FUNCTION_BLOCK XtsMotorModule EXTENDS CyclicBase IMPLEMENTS I_Initialisable, I_XtsMotorModule
VAR
	_MyModuleIoInterface : I_TcIoXtsPartModule;
	_IsInitialised : BOOL;
	CurrentLive: LREAL;
	MaxCurrent: LREAL;
	Nominal24Vdc : REAL := 24.0;
	Nominal48Vdc : REAL := 48.0;
	InSim : BOOL;
	Module24Vdc: REAL;
	Module48Vdc: REAL;
	ModuleState: Tc3_XTS_Utility.DriveState;
	ModuleStatus: Tc3_XTS_Utility.CoeStatusInfo;
	ErrorTrigger : R_TRIG;
	ModuleError: Tc3_XTS_Utility.I_AT2xxxDiagHistory;
	ReadDiagHistory: BOOL;
	ModuleDiagMessages: ARRAY [1..25] OF Tc3_XTS_Utility.ST_DiagHistoryMsg;
	NullMessage : ST_DiagHistoryMsg;
	NewDiagMessageCount : UINT;
	ModuleName: STRING;
	DriveId: Tc3_XTS_Utility.ST_DriveOnlineIdentity;
END_VAR

METHOD AckDiagMsgs : BOOL
VAR_INPUT
END_VAR
IF ModuleError = 0 THEN
	RETURN;
END_IF

ModuleError.AckAllMsgs := TRUE;
END_METHOD

METHOD PUBLIC  Cycle : HRESULT
VAR_INPUT
END_VAR
VAR
	i : INT;
END_VAR
IF _MyModuleIoInterface = 0 THEN
	Cycle := -1;
	RETURN;
END_IF

IF InSim THEN
	Cycle := -2;
	RETURN;
END_IF

CurrentLive:= _MyModuleIoInterface.GetOverallCurrent();
MaxCurrent:=  _MyModuleIoInterface.GetMaxOverallCurrentLast500ms();
Module24Vdc := _MyModuleIoInterface.GetAuxiliaryVoltage24V();
Module48Vdc := _MyModuleIoInterface.GetDCLinkVoltage();
ModuleState := _MyModuleIoInterface.GetDriveState();
ModuleStatus := _MyModuleIoInterface.GetDriveStatusInfo();
IF ModuleError.UnackMsgsAvailable THEN
	NewDiagMessageCount := ModuleError.UnackMsgCount;
	FOR i := 1 TO 25 DO
		ModuleDiagMessages[i] := NullMessage;
	END_FOR
	ModuleDiagMessages := ModuleError.DiagHistory.aDiagHistoryMsg;
END_IF

ErrorTrigger(CLK := ModuleState = DriveState.Fault OR ModuleState = DriveState.FaultReactionActive);
IF ErrorTrigger.Q OR ReadDiagHistory THEN
	ReadDiagHistory := TRUE;
	if ModuleError.UpdateDiagHistory() THEN
		ReadDiagHistory := FALSE;
	END_IF
END_IF
END_METHOD

METHOD GetLatestDiagMessage : UDINT
VAR_INPUT
END_VAR
GetLatestDiagMessage := ModuleDiagMessages[1].wDiagMessageCode;
END_METHOD

METHOD Initialise : HRESULT
VAR_INPUT
END_VAR
IF NOT _MyModuleIoInterface.P_IsInitialized THEN
	Initialise := -1;
	RETURN;
END_IF

ModuleError := _MyModuleIoInterface.CoE.DiagHistoryData;
ReadDiagHistory := TRUE;
ModuleName := _MyModuleIoInterface.P_ObjectName;
DriveId := _MyModuleIoInterface.GetDriveOnlineIdentity();
_IsInitialised := TRUE;
END_METHOD

PROPERTY Initialised : BOOL
GET
Initialised := _IsInitialised;
END_GET
END_PROPERTY

METHOD Is24VOK : HRESULT
VAR_INPUT
END_VAR
Is24VOK := 1;
IF Module24Vdc < (Nominal24Vdc * 0.8) THEN
	Is24VOK := -1;
END_IF
IF Module24Vdc > (Nominal24Vdc * 1.2) THEN
	Is24VOK := -1;
END_IF
END_METHOD

METHOD Is48VOK : HRESULT
VAR_INPUT
END_VAR
Is48VOK := 1;
IF Module48Vdc < (Nominal48Vdc * 0.9) THEN
	Is48VOK := -1;
END_IF
IF Module48Vdc > (Nominal48Vdc * 1.1) THEN
	Is48VOK := -1;
END_IF
END_METHOD

PROPERTY MyModuleInterface : I_TcIoXtsPartModule
GET
MyModuleInterface := _MyModuleIoInterface;
END_GET
SET
_MyModuleIoInterface := MyModuleInterface;
END_SET
END_PROPERTY

METHOD SetInSim : HRESULT
VAR_INPUT
END_VAR
InSim := true;
END_METHOD

END_FUNCTION_BLOCK

(* stored: Version 1.1.0.1
   POU XtsMotorModule: Id {447db564-ab24-433c-b078-4cedd1c7411e}, SpecialFunc None
   Method AckDiagMsgs: Id {d8ef1bd0-5cfc-41d5-b153-4987f2146f4f}
   Method Cycle: Id {1188f197-bbd0-4970-903a-af249f1ed9e0}
   Method GetLatestDiagMessage: Id {c5f72fde-7f4b-4c41-8777-bc94a2aa888f}
   Method Initialise: Id {0d230f78-299f-458d-bcac-a537a1290197}
   Property Initialised: Id {5149f147-92a6-4662-be65-a10eccccf631}
   Get Get: Id {7ce6f34a-06d5-4124-9539-f315dce97e7b}
   Method Is24VOK: Id {9b08696d-e0e1-46f9-950f-7b12a84e7180}
   Method Is48VOK: Id {f76f25e2-8796-412c-b16e-72d1b643b91d}
   Property MyModuleInterface: Id {2168d719-80a8-412e-a875-7c102bb8a0d2}
   Get Get: Id {89cf633f-414b-41a7-b6da-6e0666d662cd}
   Set Set: Id {c9ca3467-a5fd-4003-89ce-a9baa660bd96}
   Method SetInSim: Id {13eee03f-0b41-4595-95d5-55a5ef2b6f3f} *)
